Staubli VAL3: NCVetor.pgx

program NCVetor(trsf x_trFrame, trsf& x_trNC)
  local trsf l_trTrsf
begin


//  x_trFrame.x=x_trFrame.y=x_trFrame.z=0
//
//  //l_trTrsf=x_trFrame*{0,0,0,180,0,180}*{0,0,0,x_trNC.rx,x_trNC.ry,x_trNC.rz}
//  //l_trTrsf=!x_trFrame*l_trTrsf
//
//  l_trTrsf={0,0,0,180,0,180}*{0,0,0,x_trNC.rx,x_trNC.ry,x_trNC.rz}




//  x_trNC.rx=l_trTrsf.rx
//  x_trNC.ry=l_trTrsf.ry
//  x_trNC.rz=l_trTrsf.rz


end
